{attribute 'linkalways'} 
{attribute 'no_explicit_call' := 'This FB is a CLASS and must be accessed using methods or properties'}
{attribute 'enable_dynamic_creation'}
FUNCTION_BLOCK Node_F_VN_MaxElementElementwise_TcVnPoint2_REAL EXTENDS VisionNode
VAR
    ipContainer : _ITcVnContainer;
    aMax : _TcVnPoint2_REAL;
    hrPrev : _HRESULT(S_OK);
    hresult : _HRESULT(S_OK);
END_VAR

METHOD PUBLIC  Clone : I_Node
VAR
	pNode : POINTER TO Node_F_VN_MaxElementElementwise_TcVnPoint2_REAL;
END_VAR
pNode := __NEW(Node_F_VN_MaxElementElementwise_TcVnPoint2_REAL);
Clone := pNode^;
END_METHOD

METHOD FB_init : BOOL
VAR_INPUT
	bInitRetains : BOOL; // if TRUE, the retain variables are initialized (warm start / cold start)
	bInCopyCode : BOOL;  // if TRUE, the instance afterwards gets moved into the copy code (online change)
END_VAR
AddInput('ipContainer', ipContainer);
AddInput('hrPrev', hrPrev);
AddOutput('ipContainer', ipContainer);
AddOutput('aMax', aMax);
AddOutput('hresult',hresult);
END_METHOD

METHOD PROTECTED OnExecute
hresult.Value := F_VN_MaxElementElementwise_TcVnPoint2_REAL(
    ipContainer := ipContainer.Value,
    aMax := aMax.Value,
    hrPrev:= hrPrev.Value);
END_METHOD

METHOD PUBLIC PreExecutionCheck
VAR_INPUT
	Check : I_PreExecutionChecks;
END_VAR
Check.IsTrue(ipContainer.IsValid, 'ipContainer must be a valid container');
Check.IsTrue(ipContainer.IsType(TC_GLOBAL_CONST_LIST.ContainerType_Vector_TcVnPoint2_REAL), 'ipContainer contains incorrect type');
END_METHOD

END_FUNCTION_BLOCK

(* stored: Version 1.1.0.1, ProductVersion 3.1.4026.13
   POU Node_F_VN_MaxElementElementwise_TcVnPoint2_REAL: Id {0afcad21-d3ca-44ce-9c75-a8bfe02dce08}, SpecialFunc None
   Folder Constructor: Id {9f08a37a-17aa-4807-99a9-bcf3f0f0e2b3}
   Method Clone: Id {b9a39b4a-cc66-461a-a918-c4ac398dbb1a}
   Method FB_init: Id {7b7af533-5b07-4773-8cbc-cd3b0cf4cfb2}
   Method OnExecute: Id {c77c5a6c-6f04-4df1-a8f0-9a98aed6bb4a}
   Method PreExecutionCheck: Id {f92c121b-3147-4836-988f-d5e50ac0cc14} *)
